RESOURCE_TYPE RMT_RES (* Resource for Remote Device Management *)
  (* Standard: 61499 ITA; Description: Resource for Remote Device Management *)
  (* Version 0.1, 2007-10-10, JHC, Holobloc Inc, Moved to fb.rt. *)
  (* Version 0.0, 2001-01-08, JHC, Rockwell Automation *)
  (* Compiler header: package fb.rt; *)
  (* Compiler Java IBM VisualAge 3.0 *)
  VAR_INPUT
    MGR_ID : WSTRING := "localhost:61499"; (* Device manager socket ID *)
  END_VAR
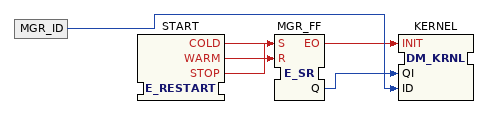
  FBS
    START : E_RESTART;
    MGR_FF : E_SR;
    KERNEL : DM_KRNL;
  END_FBS
  EVENT_CONNECTIONS
    START.COLD TO MGR_FF.S;
    START.WARM TO MGR_FF.S;
    START.STOP TO MGR_FF.R;
    MGR_FF.EO TO KERNEL.INIT;
  END_CONNECTIONS
  DATA_CONNECTIONS
    MGR_FF.Q TO KERNEL.QI;
    MGR_ID TO KERNEL.ID;
  END_CONNECTIONS
END_RESOURCE_TYPE
